// TIA Portal V21 export
FUNCTION_BLOCK "FB614"   // FB614, LAD
TITLE = FB614
{ S7_Optimized_Access := 'TRUE' }
// CIP FSC PUMP
// stored: AutoNumber false, MemoryReserve 100, SetENOAutomatically false
   VAR_INPUT
      Simulation : Bool;
      Running : Bool;
      OnCondition : Bool;
      FscInput : Bool;
      BypassFscLogic : Bool;
      OnDelay : Int;
      OffDelay : Int;
      CasingDrainDelay : Int;
   END_VAR
   VAR_OUTPUT
      Output : Bool;
      CasingDrainValve : Bool;
   END_VAR
   VAR_IN_OUT
      Temp1 : DInt;
      Temp2 : DInt;
      Temp3 : Bool;
      Temp4 : Bool;
      Temp5 : DInt;
   END_VAR
   VAR
      OnDelayTimer { S7_SetPoint := 'True'} : TON_TIME;
      BypassFSLogicForcefully { S7_SetPoint := 'True'} : TON_TIME;
      OffDelayTimer { S7_SetPoint := 'True'} : TON_TIME;
      CdTimer { S7_SetPoint := 'True'} : TON_TIME;
   END_VAR
   VAR_TEMP   // added for the SCL form of the ladder/FBD networks
      _w1 : Bool;
   END_VAR
BEGIN

REGION Network 1
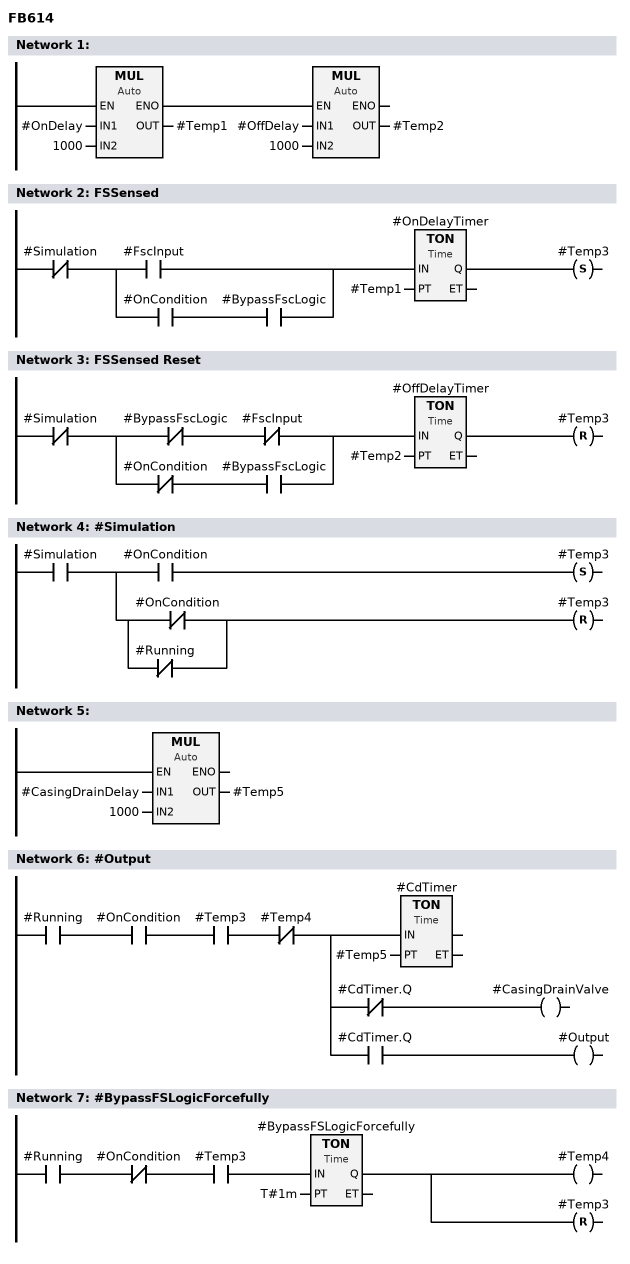
   RUNG wire#powerrail
      Mul(in1 := #OnDelay, in2 := 1000, out => #Temp1)
      Mul(in1 := #OffDelay, in2 := 1000, out => #Temp2)
   END_RUNG
   // the same network as SCL:
   #Temp1 := #OnDelay * 1000;
   #Temp2 := #OffDelay * 1000;
END_REGION

REGION Network 2: FSSensed
   RUNG wire#powerrail
      I_Contact( #Simulation )
      wire#w1
      Contact( #FscInput )
      wire#w2
      { S7_Templates := "time_type := Time" } #OnDelayTimer.TON(pt := #Temp1, et =>)
      S_Coil( #Temp3 )
   END_RUNG
   RUNG wire#w1
      Contact( #OnCondition )
      Contact( #BypassFscLogic )
   END_RUNG wire#w2
   // the same network as SCL:
   #OnDelayTimer(IN := NOT #Simulation AND (#FscInput OR (#OnCondition AND #BypassFscLogic)), PT := #Temp1);   // TON
   IF #OnDelayTimer.Q THEN #Temp3 := TRUE; END_IF;
END_REGION

REGION Network 3: FSSensed Reset
   RUNG wire#powerrail
      I_Contact( #Simulation )
      wire#w1
      I_Contact( #BypassFscLogic )
      I_Contact( #FscInput )
      wire#w2
      { S7_Templates := "time_type := Time" } #OffDelayTimer.TON(pt := #Temp2, et =>)
      R_Coil( #Temp3 )
   END_RUNG
   RUNG wire#w1
      I_Contact( #OnCondition )
      Contact( #BypassFscLogic )
   END_RUNG wire#w2
   // the same network as SCL:
   #OffDelayTimer(IN := NOT #Simulation AND ((NOT #BypassFscLogic AND NOT #FscInput) OR (NOT #OnCondition AND #BypassFscLogic)),   // TON
                  PT := #Temp2);
   IF #OffDelayTimer.Q THEN #Temp3 := FALSE; END_IF;
END_REGION

REGION Network 4: #Simulation
   RUNG wire#powerrail
      Contact( #Simulation )
      wire#w1
      Contact( #OnCondition )
      S_Coil( #Temp3 )
   END_RUNG
   RUNG wire#w1
      I_Contact( #OnCondition )
      wire#w2
      R_Coil( #Temp3 )
   END_RUNG
   RUNG wire#w1
      I_Contact( #Running )
   END_RUNG wire#w2
   // the same network as SCL:
   IF #Simulation AND #OnCondition THEN #Temp3 := TRUE; END_IF;
   IF #Simulation AND (NOT #OnCondition OR NOT #Running) THEN #Temp3 := FALSE; END_IF;
END_REGION

REGION Network 5
   RUNG wire#powerrail
      Mul(in1 := #CasingDrainDelay, in2 := 1000, out => #Temp5)
   END_RUNG
   // the same network as SCL:
   #Temp5 := #CasingDrainDelay * 1000;
END_REGION

REGION Network 6: #Output
   RUNG wire#powerrail
      Contact( #Running )
      Contact( #OnCondition )
      Contact( #Temp3 )
      I_Contact( #Temp4 )
      wire#w1
      { S7_Templates := "time_type := Time" } #CdTimer.TON(pt := #Temp5, et =>)
   END_RUNG
   RUNG wire#w1
      I_Contact( #CdTimer.Q )
      Coil( #CasingDrainValve )
   END_RUNG
   RUNG wire#w1
      Contact( #CdTimer.Q )
      Coil( #Output )
   END_RUNG
   // the same network as SCL:
   #_w1 := #Running AND #OnCondition AND #Temp3 AND NOT #Temp4;
   #CdTimer(IN := #_w1, PT := #Temp5);   // TON
   #CasingDrainValve := #_w1 AND NOT #CdTimer.Q;
   #Output := #_w1 AND #CdTimer.Q;
END_REGION

REGION Network 7: #BypassFSLogicForcefully
   RUNG wire#powerrail
      Contact( #Running )
      I_Contact( #OnCondition )
      Contact( #Temp3 )
      { S7_Templates := "time_type := Time" } #BypassFSLogicForcefully.TON(pt := T#1m, et =>)
      wire#w1
      Coil( #Temp4 )
   END_RUNG
   RUNG wire#w1
      R_Coil( #Temp3 )
   END_RUNG
   // the same network as SCL:
   #BypassFSLogicForcefully(IN := #Running AND NOT #OnCondition AND #Temp3, PT := T#1m);   // TON
   #Temp4 := #BypassFSLogicForcefully.Q;
   IF #BypassFSLogicForcefully.Q THEN #Temp3 := FALSE; END_IF;
END_REGION
END_FUNCTION_BLOCK
